{attribute 'GeneratedUsingTerminal: KL2904'}
{attribute addProperty BoxType "KL2904"}
{attribute addProperty Id "Channel_1AT %Q*Channel_1D6668A90"}
{attribute addProperty CRC "2131585449"}
{attribute addProperty Size "0"}
TYPE KL2904_7F0D69A9 :
STRUCT
	{attribute addProperty Name "Channel_1"}
	Channel_1 : Channel_1D6668A9;
END_STRUCT
END_TYPE

(* stored: Version 1.2.0.0, ProductVersion 3.1.4024.9
   DUT KL2904_7F0D69A9: Id {0af1d0bd-742e-48ee-9b5f-67a55822702a} *)
